// TIA Portal V19 export
TYPE "LEXCHANGETRAY_typeSr1000ProfinetTelegram_out"
// stored: Access Published
   STRUCT
      completionClearControlBits : "LEXCHANGETRAY_typeSr1000ProfinetTelegram_completionClearControlBits";
      latchandErrorClearControlBits { S7_SetPoint := 'True'} : "LEXCHANGETRAY_typeSr1000ProfinetTelegram_latchandErrorClearControlBits";
      operationinstructionControlBits { S7_SetPoint := 'True'} : "LEXCHANGETRAY_typeSr1000ProfinetTelegram_operationinstructionControlBits";
      parameterBankNumber { S7_SetPoint := 'True'} : "LEXCHANGETRAY_typeSr1000ProfinetTelegram_parameterBankNumber";
      userData128Byte { S7_SetPoint := 'True'} : "LEXCHANGETRAY_typeSr1000ProfinetTelegram_userData128Byte";
   END_STRUCT;
END_TYPE
